// TIA Portal project "OnlineActuator" (V14)
// For Naveed sir acurium

(* hardware
DEVICE "S7-1200 station_1"  S7-1200 Station
   slot 0: "Rack_0"  S7-1200 Rack  Rack  V1.0
   slot 1: "PLC_1"  CPU 1214C DC/DC/DC  6ES7 214-1AG31-0XB0  V3.0
*)

// ===== PLC "PLC_1"  CPU 1214C DC/DC/DC =====

VAR_GLOBAL   // PLC tag table "Default tag table"
   "actuator01" AT %M0.0 : Bool;
   "actuator02" AT %M0.1 : Bool;
   "actuator03" AT %M0.2 : Bool;
   "actuator04" AT %M0.3 : Bool;
   "actuator05" AT %M0.4 : Bool;
   "actuator06" AT %M0.5 : Bool;
   "actuator07" AT %M0.6 : Bool;
   "actuator08" AT %M0.7 : Bool;
   "actuator09" AT %M1.0 : Bool;
   "actuator10" AT %M1.1 : Bool;
   "output01" AT %Q0.0 : Bool;
   "output02" AT %Q0.1 : Bool;
   "output03" AT %Q0.2 : Bool;
   "output04" AT %Q0.3 : Bool;
   "output05" AT %Q0.4 : Bool;
   "output06" AT %Q0.5 : Bool;
   "output07" AT %Q0.6 : Bool;
   "output08" AT %Q0.7 : Bool;
   "output09" AT %Q1.0 : Bool;
   "output10" AT %Q1.1 : Bool;
END_VAR

DATA_BLOCK "system"   // DB1
{ S7_Optimized_Access := 'TRUE' }
VERSION : 0.1
   VAR RETAIN
      data : String := 'sincos';
   END_VAR
BEGIN
END_DATA_BLOCK

ORGANIZATION_BLOCK "Main"   // OB1, LAD, ProgramCycle
TITLE = "Main Program Sweep (Cycle)"
{ S7_Optimized_Access := 'TRUE' }
VERSION : 0.1
   VAR_TEMP
      RetVal : Int;
   END_VAR
BEGIN

REGION Network 1
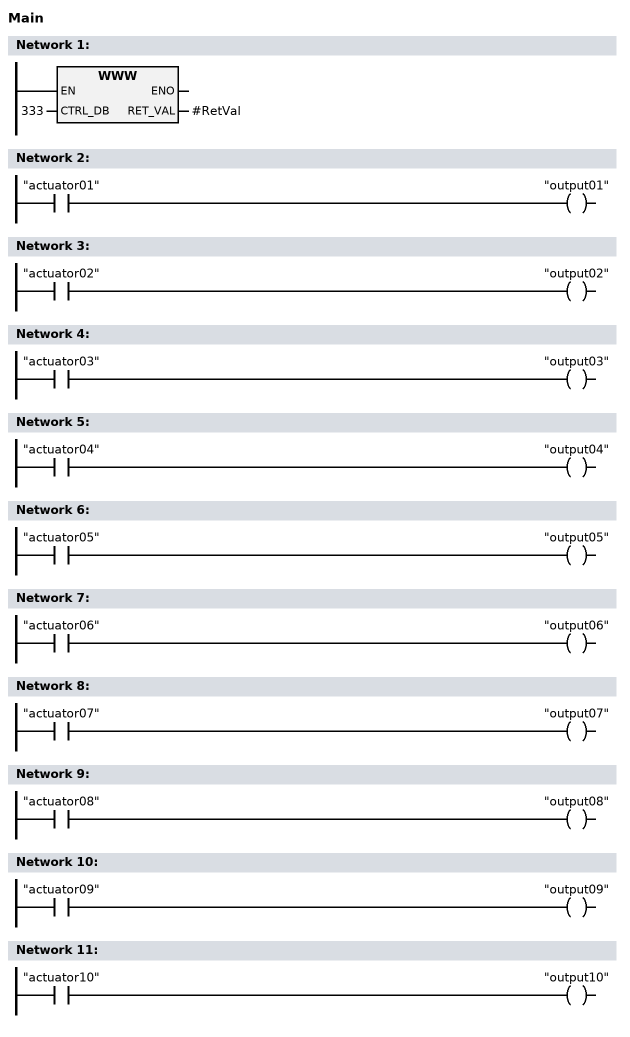
   #RetVal := WWW(CTRL_DB := 333);
END_REGION

REGION Network 2
   RUNG wire#powerrail
      Contact( "actuator01" )
      Coil( "output01" )
   END_RUNG
   // the same network as SCL:
   "output01" := "actuator01";
END_REGION

REGION Network 3
   RUNG wire#powerrail
      Contact( "actuator02" )
      Coil( "output02" )
   END_RUNG
   // the same network as SCL:
   "output02" := "actuator02";
END_REGION

REGION Network 4
   RUNG wire#powerrail
      Contact( "actuator03" )
      Coil( "output03" )
   END_RUNG
   // the same network as SCL:
   "output03" := "actuator03";
END_REGION

REGION Network 5
   RUNG wire#powerrail
      Contact( "actuator04" )
      Coil( "output04" )
   END_RUNG
   // the same network as SCL:
   "output04" := "actuator04";
END_REGION

REGION Network 6
   RUNG wire#powerrail
      Contact( "actuator05" )
      Coil( "output05" )
   END_RUNG
   // the same network as SCL:
   "output05" := "actuator05";
END_REGION

REGION Network 7
   RUNG wire#powerrail
      Contact( "actuator06" )
      Coil( "output06" )
   END_RUNG
   // the same network as SCL:
   "output06" := "actuator06";
END_REGION

REGION Network 8
   RUNG wire#powerrail
      Contact( "actuator07" )
      Coil( "output07" )
   END_RUNG
   // the same network as SCL:
   "output07" := "actuator07";
END_REGION

REGION Network 9
   RUNG wire#powerrail
      Contact( "actuator08" )
      Coil( "output08" )
   END_RUNG
   // the same network as SCL:
   "output08" := "actuator08";
END_REGION

REGION Network 10
   RUNG wire#powerrail
      Contact( "actuator09" )
      Coil( "output09" )
   END_RUNG
   // the same network as SCL:
   "output09" := "actuator09";
END_REGION

REGION Network 11
   RUNG wire#powerrail
      Contact( "actuator10" )
      Coil( "output10" )
   END_RUNG
   // the same network as SCL:
   "output10" := "actuator10";
END_REGION
END_ORGANIZATION_BLOCK